PROGRAM Kommunikation
VAR
	
	// Instanziierung der Auswertung:
	Auswertung		:FB_Auswertung;
	Mode			:FB_Modus;
	
	// Instanziierung der Grundfunktionen: 
	Entleeren		:GF_Entleeren;
	//Halten			:GF_Halten;
	Pumpen			:GF_Pumpen;
	Zirkulieren		:GF_Zirkulieren;
	Ruehren 		:GF_Ruehren;
	Warten			:GF_Warten;	
	Befuellen		:GF_Befuellen;	
	Leitung			:FB_Leitungswahl;

END_VAR

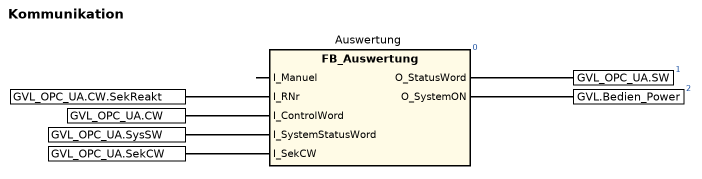
Auswertung(
    I_RNr := GVL_OPC_UA.CW.SekReakt,
    I_ControlWord := GVL_OPC_UA.CW,
    I_SystemStatusWord := GVL_OPC_UA.SysSW,
    I_SekCW := GVL_OPC_UA.SekCW); // FB_Auswertung
GVL_OPC_UA.SW := Auswertung.O_StatusWord;
GVL.Bedien_Power := Auswertung.O_SystemON;

END_PROGRAM

(* stored: Version 1.1.0.1, ProductVersion 3.1.4024.12
   POU Kommunikation: Id {36ca285f-8f18-49ff-80f3-f202fc5db8df}, SpecialFunc None *)
